PROGRAM IpcDiagnostics
VAR CONSTANT
	cNetId			: T_AmsNetID := '';				// local
	cNbrParameters	: UDINT := 8;					// number of parameters to read 
END_VAR
VAR
	bStart			: BOOL := TRUE;       			// flag to trigger (re)start of statemachine
	eState			: E_State := E_State.Init;
	hrGetValue		: HRESULT;	

	sDeviceName		: STRING(39);
	nCpuFreq		: UDINT;
	nTcBuild		: UINT;
	aNetworkNames	: ARRAY[1..3] OF STRING(79);	// array in order to receive info of up to three network ports (NICs)
	aIpAddr			: ARRAY[1..3] OF STRING(39);	// array in order to receive info of up to three network ports (NICs)
	aDHCP			: ARRAY[1..3] OF BOOL;			// array in order to receive info of up to three network ports (NICs)
	sMdpVersion		: STRING;
	nBootCnt		: UDINT;
	
	nCpuTemperature	: INT;							// [°C]; should be read periodically
	

	fbDiagRegister	: FB_IPCDiag_Register := (sNetId:=cNetId);
	fbDiagRead		: FB_IPCDiag_ReadParameter := (sNetId:=cNetId);
	nKeyIdx			: USINT := 1;
	aParameterKeys	: ARRAY[1..cNbrParameters] OF E_IPCDiag_ParameterKey := [	E_IPCDiag_ParameterKey.IPCDeviceName,
																				E_IPCDiag_ParameterKey.CPU_Frequency,
																				E_IPCDiag_ParameterKey.TC_VersionBuild,
																				E_IPCDiag_ParameterKey.NIC_Name,
																				E_IPCDiag_ParameterKey.NIC_IPv4Address,
																				E_IPCDiag_ParameterKey.NIC_DHCP,
																				E_IPCDiag_ParameterKey.Software_MDPVersion,
																				E_IPCDiag_ParameterKey.MB_BootCnt ];
	fbDiagReadPeriodic : FB_IPCDiag_ReadParameterPeriodic := (eParameterKey:=E_IPCDiag_ParameterKey.CPU_Temp, tPeriod:= T#10S, sNetId:=cNetId);
END_VAR

CASE eState OF
E_State.Init:
	IF NOT fbDiagRegister.bBusy THEN
		fbDiagRegister(bExecute:=TRUE); // need to be executed once
	ELSE
		fbDiagRegister(bExecute:=FALSE);
	END_IF
	IF NOT fbDiagRegister.bBusy THEN
		IF fbDiagRegister.bError THEN
			eState := E_State.Error;
		ELSE
			eState := E_State.Idle;
		END_IF
	END_IF

E_State.Idle:	
    IF bStart THEN
        bStart := FALSE;
        eState := E_State.ReadOnce;
    END_IF
	
E_State.ReadOnce: // reads every parameter once
	IF NOT fbDiagRead.bBusy THEN
		fbDiagRead(bExecute:= TRUE, eParameterKey:=aParameterKeys[nKeyIdx], fbRegister:=fbDiagRegister);	
	ELSE
		fbDiagRead(bExecute:= FALSE, fbRegister:=fbDiagRegister);
	END_IF
	IF NOT fbDiagRead.bBusy THEN
		IF fbDiagRead.bError THEN
			eState := E_State.Error;
		ELSE // get value
			IF aParameterKeys[nKeyIdx] = E_IPCDiag_ParameterKey.IPCDeviceName THEN
				hrGetValue := fbDiagRead.GetParameter(pBuffer:=ADR(sDeviceName), nBufferSize:=SIZEOF(sDeviceName));
				
			ELSIF aParameterKeys[nKeyIdx] = E_IPCDiag_ParameterKey.CPU_Frequency THEN
				hrGetValue := fbDiagRead.GetParameter(pBuffer:=ADR(nCpuFreq), nBufferSize:=SIZEOF(nCpuFreq));
				
			ELSIF aParameterKeys[nKeyIdx] = E_IPCDiag_ParameterKey.TC_VersionBuild THEN
				hrGetValue := fbDiagRead.GetParameter(pBuffer:=ADR(nTcBuild), nBufferSize:=SIZEOF(nTcBuild));
				
			ELSIF aParameterKeys[nKeyIdx] = E_IPCDiag_ParameterKey.NIC_Name THEN
				// get values (one by one)
				hrGetValue := fbDiagRead.GetParameterByIdx(pBuffer:=ADR(aNetworkNames[1]), nBufferSize:=SIZEOF(aNetworkNames[1]), 1);
				IF SUCCEEDED(hrGetValue) THEN
					hrGetValue := fbDiagRead.GetParameterByIdx(pBuffer:=ADR(aNetworkNames[2]), nBufferSize:=SIZEOF(aNetworkNames[2]), 2);
				END_IF				
			ELSIF aParameterKeys[nKeyIdx] = E_IPCDiag_ParameterKey.NIC_IPv4Address THEN
				// get values (all together)
				hrGetValue := fbDiagRead.GetParameterStrings(pBuffer:=ADR(aIpAddr), nBufferSize:=SIZEOF(aIpAddr), nStrings:=3);
				
			ELSIF aParameterKeys[nKeyIdx] = E_IPCDiag_ParameterKey.NIC_DHCP THEN
				// get values (all together)
				hrGetValue := fbDiagRead.GetParameter(pBuffer:=ADR(aDHCP), nBufferSize:=SIZEOF(aDHCP));
				
			ELSIF aParameterKeys[nKeyIdx] = E_IPCDiag_ParameterKey.Software_MDPVersion THEN
				hrGetValue := fbDiagRead.GetParameter(pBuffer:=ADR(sMdpVersion), nBufferSize:=SIZEOF(sMdpVersion));
			
			ELSIF aParameterKeys[nKeyIdx] = E_IPCDiag_ParameterKey.MB_BootCnt THEN
				hrGetValue := fbDiagRead.GetParameter(pBuffer:=ADR(nBootCnt), nBufferSize:=SIZEOF(nBootCnt));
			
			END_IF
				
			IF SUCCEEDED(hrGetValue) THEN
				IF nKeyIdx = cNbrParameters THEN // all keys successfully read
					nKeyIdx := 1;
					eState := E_State.ReadPeriodically;
				ELSE
					nKeyIdx := nKeyIdx + 1;
				END_IF
			ELSE
				eState := E_State.Error;
			END_IF
		END_IF
	END_IF	

E_State.ReadPeriodically:
	fbDiagReadPeriodic(bEnable:=TRUE, fbRegister:=fbDiagRegister);
	IF fbDiagReadPeriodic.bValid THEN
		fbDiagReadPeriodic.GetParameter(pBuffer:=ADR(nCpuTemperature), nBufferSize:=SIZEOF(nCpuTemperature) );	
	END_IF
	IF fbDiagReadPeriodic.bError THEN
		eState := E_State.Error;
	END_IF	
	
E_State.Error:
	(* implementation of error logging and error handling *)
	(* hint: An error could also occur if a parameter is not supported by chosen hardware or image. 
	E.g. not all IPCs offer a CPU temperature measurement. *)

END_CASE

END_PROGRAM

(* stored: Version 1.1.0.1, ProductVersion 3.1.4022.18
   POU IpcDiagnostics: Id {d4b9ca14-f27d-4d64-abbf-78404738a3dc}, SpecialFunc None *)
